Staubli VAL3: remMovBase.pgx

program remMovBase(point& pDest[] (dimensions=1), string& sReturn[] (dimensions=1))
  local bool bMovOk
  local joint jDest
  local joint jHere
  local mdesc mUserSpeed
  local num nDistance
  local string sGoal
  local trsf trGoal
begin
  // Move to a given point, handling movement
  // parameters and stay clear zones.
  //
  logMsg("call remMovBase")
  //first, check if movement is possible.
  jHere=herej()
  bMovOk=pointToJoint(tSensorTool,jHere,pDest,jDest)
  if bMovOk
    //check if we're moving too far (user set max dist)
    nDistance=abs(distance(here(tSensorTool,world),pDest))
    //put a line to say where we're going to
    trGoal=pDest.trsf
    sGoal="Moving "+toString(sNumConv,nDistance)+" mm to ("
    sGoal=sGoal+toString(sNumConv,trGoal.x)+", "
    sGoal=sGoal+toString(sNumConv,trGoal.y)+", "
    sGoal=sGoal+toString(sNumConv,trGoal.z)+", "
    sGoal=sGoal+toString(sNumConv,trGoal.rx)+", "
    sGoal=sGoal+toString(sNumConv,trGoal.ry)+", "
    sGoal=sGoal+toString(sNumConv,trGoal.rz)+")"
    putln(sGoal)
    logMsg(sGoal)
    if nDistance<nMaxDist
      mUserSpeed={nMaxAccel,100,nMaxAccel,nMaxVelo,nMaxRVelo,off,50,50}
      call iocWriteBack("ARMMOVING")
      putln("ARM MOVING")
      logMsg("ARM MOVING")
      bEnableMonitor=true
      if bMoveLinear
        movel(pDest,tSensorTool,mUserSpeed)
      else
        movej(jDest,tSensorTool,mUserSpeed)
      endIf
      //watch for stay clear zones
      do
        nDistance=abs(distance(here(tSensorTool,world),pDest))
        delay(0)
        //stop checking if done or if zone is violated
      until nDistance<=nZoneWatchTol or bInsideCube or bInsideCylinder or bInsideSphere
      //stop and raise error if we violated a stay clear zone
      if bInsideCube or bInsideCylinder or bInsideSphere
        stopMove()
        resetMotion()
        bStopAllMonitor=true
        call remErrZone(sReturn)
      else
        waitEndMove()
        sReturn=""
      endIf
      putln("ARM DONE MOVING")
      logMsg("ARM DONE MOVING")
      bEnableMonitor=false
    else
      //destination was too far, so we raise an error
      call remErrFar(sReturn)
    endIf
  else
    //destination was impossible, so we raise an error
    call remErrConfig(sReturn)
  endIf
end
